Staubli VAL3: OnEvent.dtx

string sGun[2]
  [0] = "valve1"
  [1] = "valve2"
mdesc nom_speed = {tmax=9999, rmax=9999, blend=off}
public dio valve1 = {link=valve1}
public dio valve2 = {link=valve2}
